INTERFACE IRecordDB

PROPERTY query : string(512)
GET
END_GET
SET
END_SET
END_PROPERTY

PROPERTY queue : REFERENCE TO dequeue
GET
END_GET
SET
END_SET
END_PROPERTY

END_INTERFACE

(* stored: Version 1.1.0.1, ProductVersion 3.1.4024.12
   Itf IRecordDB: Id {1d7da905-9dbc-4a62-9363-d7eaf62f12d7}
   Property query: Id {0c693f22-a1e1-4998-bbc5-28f2eaaa08a9}
   Get Get: Id {769bd1ee-8ee2-4d6a-b905-0865d7739bb5}
   Set Set: Id {b5ea8c81-b164-4a8f-a1cc-84f0e1214dde}
   Property queue: Id {18d54e9e-17bd-4a1e-8024-4a0247b3ade1}
   Get Get: Id {d1e55aac-b05f-4975-8355-8cb725db3b42}
   Set Set: Id {31f7b075-694c-4eea-b938-0dbf3bc2b8ab} *)
